FUNCTION_BLOCK FB_HeatPumpSystem EXTENDS FB_SystemContinous
VAR_INPUT
END_VAR
VAR_OUTPUT
END_VAR
VAR
	//Vitocal 350-G heat pump
	HeatPump : FB_HeatPump;
	
	//valve 146 and valve 246
	ST_SV146DefaultParameters : ST_DiscreteValveDefaultParameters := (bFeedbackSignal := FALSE);
	ST_SV246DefaultParameters : ST_DiscreteValveDefaultParameters := (bFeedbackSignal := FALSE);	
	SV146 : FB_DiscreteValve := (ST_DefaultParameters := ST_SV146DefaultParameters);
	SV246 : FB_DiscreteValve := (ST_DefaultParameters := ST_SV246DefaultParameters);	
	
	//internal variables
	bSetStatusOn_HeatPump : BOOL;
	bSetStatusOn_SV146 : BOOL;
	bSetStatusOn_SV246 : BOOL;
	
	bStartTimer : BOOL;
	Timer : TON;
END_VAR

MAIN();
//use timer because valve has no feedback signal (75 sec)
Timer(IN := bStartTimer,
	PT := T#75S);

//heat pump
HeatPump(bSetStatusOnAutomatic := bSetStatusOn_HeatPump,
	bAlgorithmPermission := bAlgorithmPermission);
HeatPump.SetState_BO();

//valves
SV146(bSetStatusOnAutomatic := bSetStatusOn_SV146,
		bAlgorithmPermission := bAlgorithmPermission);
SV146.SetState_BI_BO();
		
SV246(bSetStatusOnAutomatic := bSetStatusOn_SV246,
		bAlgorithmPermission := bAlgorithmPermission);
SV246.SetState_BI_BO();

METHOD PROTECTED  CheckError : BOOL
VAR_INPUT
END_VAR
VAR_OUTPUT
	bError : BOOL;
END_VAR
//empty method because system has no feedback signals
END_METHOD

METHOD PROTECTED  Operational : BOOL
VAR_INPUT
END_VAR
VAR_OUTPUT
	bSwitchToWorking : BOOL := FALSE;
END_VAR
bSetStatusOn_HeatPump := TRUE;
bSwitchToWorking := TRUE;
END_METHOD

METHOD PROTECTED  RampDown : BOOL
VAR_INPUT
END_VAR
VAR_OUTPUT
	bRampDownFinished : BOOL := FALSE;
END_VAR
bSetStatusOn_HeatPump := FALSE;
bSetStatusOn_SV146 := FALSE;
bSetStatusOn_SV246 := FALSE;
bStartTimer := TRUE;

IF Timer.Q THEN
	bRampDownFinished := TRUE;
	bStartTimer := FALSE;
END_IF
END_METHOD

METHOD PROTECTED  RampUp : BOOL
VAR_INPUT
END_VAR
VAR_OUTPUT
	bRampUpFinished : BOOL := FALSE;
END_VAR
bSetStatusOn_SV146 := TRUE;
bSetStatusOn_SV246 := TRUE;
bStartTimer := TRUE;

IF Timer.Q THEN
	bRampUpFinished := TRUE;
	bStartTimer := FALSE; //resets timer
END_IF
END_METHOD

METHOD PROTECTED   SetSetPointLimits : BOOL
VAR_INPUT
END_VAR
//heat pump has no continous setpoint (limits are not used) but must be implemented because of abstract method
aSetPointLimits[1] := 0;
aSetPointLimits[2] := 100;
END_METHOD

METHOD PROTECTED  Working : BOOL
VAR_INPUT
END_VAR
VAR_OUTPUT
	bSwitchToOperational : BOOL := FALSE;
END_VAR
//empty method because setpoint does not change during operation
END_METHOD

END_FUNCTION_BLOCK

(* stored: Version 1.1.0.1, ProductVersion 3.1.4024.10
   POU FB_HeatPumpSystem: Id {7e7b5d95-fc91-49dd-b95e-a9f45915aabb}, SpecialFunc None
   Method CheckError: Id {e6a4ede8-dc18-488e-9b82-544068cf9d4e}
   Method Operational: Id {5647c897-a33a-44f7-bde1-edb8a50b8012}
   Method RampDown: Id {1da118c0-c5a3-4c43-b5c2-92112ab088e3}
   Method RampUp: Id {18497967-281e-48be-9d5b-3e53109a49a9}
   Method SetSetPointLimits: Id {76f57d3d-d47f-4242-8b02-e8c62a723fc1}
   Method Working: Id {80b089c4-4cdc-43e9-85f7-5ded4d853262} *)
